// TIA Portal V17 export
// export: Created 2026-05-13T16:54:41.7509124Z, ExportSetting WithDefaults, DisplayName Totally Integrated Automation Portal, DisplayVersion V17 Update 4, DisplayName TIA Portal Openness, DisplayVersion V17 Update 4, DisplayName TIA Portal Version Control Interface, DisplayVersion V17, DisplayName SINAMICS Startdrive Advanced, DisplayVersion V17, DisplayName SINAMICS Startdrive G130, G150, S120, S150, SINAMICS MV, S210, DisplayVersion V17, DisplayName SINAMICS Startdrive G110M, G120, G120C, G120D, G120P, G115D, DisplayVersion V17, DisplayName STEP 7 Professional, DisplayVersion V17 Update 4, DisplayName STEP 7 Safety, DisplayVersion V17, DisplayName WinCC Professional, DisplayVersion V17 Update 4
TagTable "YB"
  YB_读重量 : Real  (PLC tag YB.读重量, HMI_连接_1, 1 s)
  YB_A瞬时流量 : Real  (PLC tag YB.A瞬时流量, HMI_连接_1, 1 s)
  YB_A瞬时流速 : Real  (PLC tag YB.A瞬时流速, HMI_连接_1, 1 s)
  YB_A介质温度 : Real  (PLC tag YB.A介质温度, HMI_连接_1, 1 s)
  YB_A当前电流 : Real  (PLC tag YB.A当前电流, HMI_连接_1, 1 s)
  YB_A流速下限 : Real  (PLC tag YB.A流速下限, HMI_连接_1, 1 s)
  YB_A流速上限 : Real  (PLC tag YB.A流速上限, HMI_连接_1, 1 s)
  YB_A管道内径 : Real  (PLC tag YB.A管道内径, HMI_连接_1, 1 s)
  YB_B瞬时流量 : Real  (PLC tag YB.B瞬时流量, HMI_连接_1, 1 s)
  YB_B瞬时流速 : Real  (PLC tag YB.B瞬时流速, HMI_连接_1, 1 s)
  YB_B介质温度 : Real  (PLC tag YB.B介质温度, HMI_连接_1, 1 s)
  YB_B当前电流 : Real  (PLC tag YB.B当前电流, HMI_连接_1, 1 s)
  YB_B流速下限 : Real  (PLC tag YB.B流速下限, HMI_连接_1, 1 s)
  YB_B流速上限 : Real  (PLC tag YB.B流速上限, HMI_连接_1, 1 s)
  YB_B管道内径 : Real  (PLC tag YB.B管道内径, HMI_连接_1, 1 s)
  YB_秤状态 : Array [0..15] of Bool  (PLC tag YB.秤状态, HMI_连接_1, 1 s)
    TagArrayMember "[0]"
    TagArrayMember "[1]"
    TagArrayMember "[2]"
    TagArrayMember "[3]"
    TagArrayMember "[4]"
    TagArrayMember "[5]"
    TagArrayMember "[6]"
    TagArrayMember "[7]"
    TagArrayMember "[8]"
    TagArrayMember "[9]"
    TagArrayMember "[10]"
    TagArrayMember "[11]"
    TagArrayMember "[12]"
    TagArrayMember "[13]"
    TagArrayMember "[14]"
    TagArrayMember "[15]"
  YB_秤操作 : Array [0..2] of Bool  (PLC tag YB.秤操作, HMI_连接_1, 1 s)
    TagArrayMember "[0]"
    TagArrayMember "[1]"
    TagArrayMember "[2]"
